{attribute 'linkalways'} 
{attribute 'no_explicit_call' := 'This FB is a CLASS and must be accessed using methods or properties'}
{attribute 'enable_dynamic_creation'}
FUNCTION_BLOCK _TcVnVector3_SINT EXTENDS AliasDatatypeBase
VAR
	localData : TcVnVector3_SINT;
	activeData : REFERENCE TO TcVnVector3_SINT REF= localData;
	aliasBaseDatatype : _Array0to2OfSINT;
END_VAR

PROPERTY PUBLIC Address : PVOID
GET
Address := ADR(activeData);
END_GET
END_PROPERTY

METHOD PUBLIC ClearReference
VAR_INPUT
END_VAR
activeData REF= localData;
SetBaseDatatypeReference();
END_METHOD

METHOD PUBLIC Clone : I_Datatype
VAR
    pClone : POINTER TO _TcVnVector3_SINT;
END_VAR
pClone := __NEW(_TcVnVector3_SINT);
Clone := pClone^;
END_METHOD

METHOD FB_init : BOOL
VAR_INPUT
	bInitRetains : BOOL; // if TRUE, the retain variables are initialized (warm start / cold start)
	bInCopyCode : BOOL;  // if TRUE, the instance afterwards gets moved into the copy code (online change)
	//InitialValue : <type>; // if possible, not all values can be initialized
END_VAR
//localData := InitialValue; // if possible, not all values can be initialized
SetBaseDatatypeReference();
AddBaseDatatype(aliasBaseDatatype);
END_METHOD

PROPERTY PUBLIC Identifier : T_MAXSTRING
GET
Identifier := 'TcVnVector3_SINT';
END_GET
END_PROPERTY

METHOD PUBLIC MakeReferenceTo
VAR_INPUT
	ReferenceTarget : REFERENCE TO TcVnVector3_SINT;
END_VAR
activeData REF= ReferenceTarget;
SetBaseDatatypeReference();
END_METHOD

METHOD PROTECTED SetBaseDatatypeReference
VAR_INPUT
END_VAR
aliasBaseDatatype.MakeReferenceTo(activeData);
END_METHOD

PROPERTY PUBLIC Size : UDINT
GET
Size := SIZEOF(activeData);
END_GET
END_PROPERTY

METHOD TryMakeReferenceTo : BOOL
VAR_INPUT
	Target : I_Datatype;
END_VAR
VAR
	pTargetData : POINTER TO TcVnVector3_SINT;
END_VAR
IF NOT IsEquivalentTo(Target) THEN
	RETURN;
END_IF

pTargetData := Target.Address;
activeData REF= pTargetData^;
SetBaseDatatypeReference();
TryMakeReferenceTo := TRUE;
END_METHOD

PROPERTY PUBLIC Value : REFERENCE TO TcVnVector3_SINT
GET
Value REF= activeData;
END_GET
END_PROPERTY

END_FUNCTION_BLOCK

(* stored: Version 1.1.0.1, ProductVersion 3.1.4024.13
   POU _TcVnVector3_SINT: Id {30485021-c03b-0223-08c3-2e60bca60873}, SpecialFunc None
   Folder Core: Id {7e874b8c-c62a-0e5a-0dc7-f7915cf54b76}
   Folder Protected: Id {92957d75-4346-0979-1589-1e1ed0e0d9f5}
   Folder Customize: Id {1ecedc4d-82fc-09f6-14be-f26868dd6ff5}
   Folder Constructor: Id {c5ba7bab-7dcc-04fc-006f-d1f7118756b6}
   Property Address: Id {45466878-28d3-0143-1f96-8b6f9bee0719}
   Get Get: Id {768ea05f-94ce-0ae2-13fb-f1ede620c78a}
   Method ClearReference: Id {36d6352f-3090-07e0-2289-11ac94aaeb8c}
   Method Clone: Id {fbf675ef-2c0c-001b-2dce-eda711c7037a}
   Method FB_init: Id {a37c66bc-0c04-0f2f-13bf-c5701cb25082}
   Property Identifier: Id {1ff214e4-508d-0917-05f7-df92027a6058}
   Get Get: Id {7f2b2a30-eb99-07d6-09d2-1f9b8c05fe81}
   Method MakeReferenceTo: Id {8a5ad0fc-55c3-073e-3445-4af13350b947}
   Method SetBaseDatatypeReference: Id {ab132ed6-266f-03af-20c5-8f3472c1904e}
   Property Size: Id {47edd0ca-9667-087c-21b1-9045a3647d9b}
   Get Get: Id {682f59ef-b8f5-0b81-0710-f6bf7c657ec6}
   Method TryMakeReferenceTo: Id {263c86c2-75c9-0734-0b32-10016b14bdda}
   Property Value: Id {21d3009e-8442-03d1-00e6-f48c00c94435}
   Get Get: Id {c421ba02-e9fa-0438-1f86-2ba694cc95d0} *)
